FUNCTION_BLOCK DualHysteresis_AR_A2X (* 2-way conversion of Analog to Digital with Hysteresis (Switch-on = MI +/- (ABS(DEAD) + ABS(HYSTERESIS)), Switch-off = MI +/- ABS(DEAD)), UP/DOWN output on a single A2X adapter *)
  (* Standard: 61499-2; Description: Copyright (c) 2026 HR Agrartechnik GmbH This program and the accompanying materials are made available under the terms of the Eclipse Public License 2.0 which is available at https://www.eclipse.org/legal/epl-2.0/ SPDX-License-Identifier: EPL-2.0 *)
  (* Version 1.0, 2026-09-05, Franz Höpfinger, HR Agrartechnik GmbH, initial API and implementation and/or initial documentation *)
  PACKAGE logiBUS::signalprocessing::hysteresis;
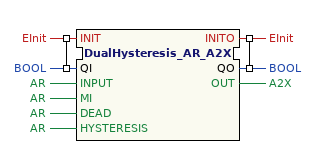
  EVENT_INPUT
    INIT : EInit WITH QI; (* Initialization Request *)
  END_EVENT
  EVENT_OUTPUT
    INITO : EInit WITH QO; (* Initialization Confirm *)
  END_EVENT
  VAR_INPUT
    QI : BOOL; (* Input event qualifier *)
  END_VAR
  VAR_OUTPUT
    QO : BOOL;
  END_VAR
  SOCKETS
    INPUT : adapter::types::unidirectional::AR; (* Input value *)
    MI : adapter::types::unidirectional::AR; (* Center point (e.g. 0.5 for 50%) *)
    DEAD : adapter::types::unidirectional::AR; (* Deadband around MI (absolute value). Switch-off points = MI +/- ABS(DEAD) *)
    HYSTERESIS : adapter::types::unidirectional::AR; (* Hysteresis value (absolute value). Switch-on points = MI +/- (ABS(DEAD) + ABS(HYSTERESIS)) *)
  END_SOCKETS
  PLUGS
    OUT : adapter::types::unidirectional::A2X; (* UP/DOWN output *)
  END_PLUGS
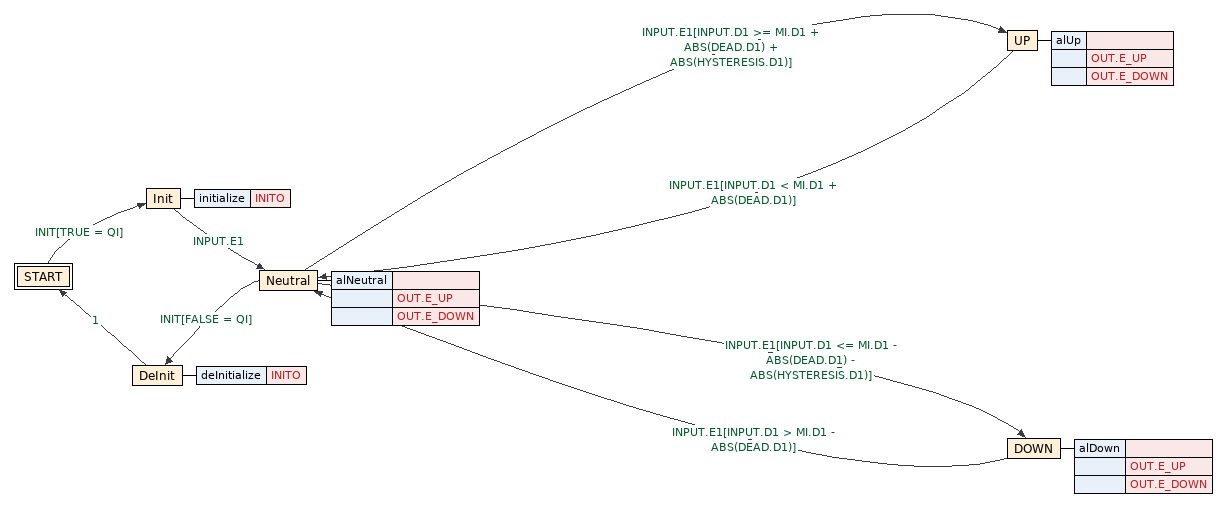
  EC_STATES
    START; (* Initial State *)
    Init : initialize -> INITO; (* Initialization *)
    UP : alUp, -> OUT.E_UP, -> OUT.E_DOWN; (* Normal execution *)
    Neutral : alNeutral, -> OUT.E_UP, -> OUT.E_DOWN;
    DeInit : deInitialize -> INITO;
    DOWN : alDown, -> OUT.E_UP, -> OUT.E_DOWN;
  END_STATES
  EC_TRANSITIONS
    START TO Init := INIT[TRUE = QI];
    Init TO Neutral := INPUT.E1;
    Neutral TO DeInit := INIT[FALSE = QI];
    Neutral TO UP := INPUT.E1[INPUT.D1 >= MI.D1 + ABS(DEAD.D1) + ABS(HYSTERESIS.D1)]; (* Switch-on UP (inclusive) *)
    DeInit TO START := 1;
    Neutral TO DOWN := INPUT.E1[INPUT.D1 <= MI.D1 - ABS(DEAD.D1) - ABS(HYSTERESIS.D1)]; (* Switch-on DOWN (inclusive) *)
    DOWN TO Neutral := INPUT.E1[INPUT.D1 > MI.D1 - ABS(DEAD.D1)]; (* Switch-off DOWN (strict) *)
    UP TO Neutral := INPUT.E1[INPUT.D1 < MI.D1 + ABS(DEAD.D1)]; (* Switch-off UP (strict) *)
  END_TRANSITIONS
  ALGORITHM initialize IN ST:
QO := QI;
(* in any case go safe State *)
OUT.UP := BOOL#FALSE;
OUT.DOWN := BOOL#FALSE;
  END_ALGORITHM
  ALGORITHM deInitialize IN ST:
QO := BOOL#FALSE;
(* in any case go safe State *)
OUT.UP := BOOL#FALSE;
OUT.DOWN := BOOL#FALSE;
  END_ALGORITHM
  ALGORITHM alNeutral IN ST:
QO := QI;
(* in any case go safe State *)
OUT.UP := BOOL#FALSE;
OUT.DOWN := BOOL#FALSE;
  END_ALGORITHM
  ALGORITHM alUp IN ST:
QO := QI;
IF TRUE = QI THEN
	(* only perform normal operation of QI is true *)
	OUT.UP := BOOL#TRUE;
	OUT.DOWN := BOOL#FALSE;
END_IF;
  END_ALGORITHM
  ALGORITHM alDown IN ST:
QO := QI;
IF TRUE = QI THEN
	(* only perform normal operation of QI is true *)
	OUT.UP := BOOL#FALSE;
	OUT.DOWN := BOOL#TRUE;
END_IF;
  END_ALGORITHM
END_FUNCTION_BLOCK
